
// ===== library types =====

// folder: NN_types

TYPE "scaler_type"
   STRUCT
      data_min : Array[1.."MAX_NO_NEURONS_PER_LAYER"] of Real;
      data_max : Array[1.."MAX_NO_NEURONS_PER_LAYER"] of Real;
      range_min : Real;
      range_max : Real;
   END_STRUCT;
END_TYPE

TYPE "NN_config_type"
   STRUCT
      NumLayers : Int := 5;
      NeuronPerLayer : Array[1.."MAX_NO_LAYERS"] of Int;
      ActivationFunction : Array[1.."MAX_NO_LAYERS"] of Int;   // 1=sigmoid; 2=ReLU; 3= Tanh; 4=LeakyReLU; 5= Softmax
      neuron : Array[1.."MAX_NO_LAYERS", 1.."MAX_NO_NEURONS_PER_LAYER"] of Real;
      weight : Array[1.."MAX_NO_LAYERS", 1.."MAX_NO_NEURONS_PER_LAYER", 1.."MAX_NO_NEURONS_PER_LAYER"] of Real;
      bias : Array[1.."MAX_NO_LAYERS", 1.."MAX_NO_NEURONS_PER_LAYER"] of Real;
      scalerParam : "scaler_type";
   END_STRUCT;
   // NeuronPerLayer[1] := 7;
   // NeuronPerLayer[2] := 128;
   // NeuronPerLayer[3] := 64;
   // NeuronPerLayer[4] := 32;
   // NeuronPerLayer[5] := 6;
   // ActivationFunction[1] := 2;
   // ActivationFunction[2] := 2;
   // ActivationFunction[3] := 2;
   // ActivationFunction[4] := 2;
   // ActivationFunction[5] := 5;
END_TYPE

// folder: NN

FUNCTION_BLOCK "NN_MLP"   // FB19000, SCL
{ S7_Optimized_Access := 'TRUE' }
VERSION : 0.1
   VAR_INPUT
      predict : Bool;
      contPredict : Bool;
      X : Array[1.."MAX_NO_NEURONS_PER_LAYER"] of Real;
   END_VAR
   VAR_OUTPUT
      done : Bool;
      busy : Bool;
      probability : Array[1.."MAX_NO_NEURONS_PER_LAYER"] of Real;
   END_VAR
   VAR_IN_OUT
      config : "NN_config_type";
   END_VAR
   VAR
      X_scaled : Array[1.."MAX_NO_NEURONS_PER_LAYER"] of Real;
      p : Int;
      n : Int;
      neuron_L : Int;
      "neuron_L+1" : Int;
      k : Int;
      layer_L : Int;
      s1 : Int;
      s2 : Int;
      S3 : Int;
      S4 : Int;
      statSumEXP : Real;
      statEXP : Array[1..6] of Real;
      statSoftmax : Array[1..6] of Real;
      statTotalSum : Real;
      predictRT : R_TRIG;
      statMemRuntime : LReal;
      timeExecution : LReal;
   END_VAR
BEGIN
   #predictRT(CLK := #predict);
   IF #predictRT.Q OR #contPredict THEN
       #timeExecution:= RUNTIME(#statMemRuntime);

       #done := FALSE;
       #busy := TRUE;

       REGION Entradas dos dados do processo  
           // normalização dos valores de entrada da rede neural. Dados retirados da função MinMaxScaler utilizada no tratamento dos dados da aplicação em python
           #config.scalerParam.data_min[1] := 295.3;
           #config.scalerParam.data_min[2] := 305.7;
           #config.scalerParam.data_min[3] := 1168.0;
           #config.scalerParam.data_min[4] := 3.8;
           #config.scalerParam.data_min[5] := 0.0;
           #config.scalerParam.data_min[6] := 0.0;
           #config.scalerParam.data_min[7] := 0.0;

           #config.scalerParam.data_max[1] := 304.5;
           #config.scalerParam.data_max[2] := 313.8;
           #config.scalerParam.data_max[3] := 2886.0;
           #config.scalerParam.data_max[4] := 76.6;
           #config.scalerParam.data_max[5] := 253.0;
           #config.scalerParam.data_max[6] := 1.0;
           #config.scalerParam.data_max[7] := 1.0;

           #config.scalerParam.range_min := -1.0;
           #config.scalerParam.range_max := 1.0;

           FOR #n := 1 TO #config.NeuronPerLayer[1] DO
               #X_scaled[#n] := (#X[#n] - #config.scalerParam.data_min[#n]) /
               (#config.scalerParam.data_max[#n] - #config.scalerParam.data_min[#n]) *
               (#config.scalerParam.range_max - #config.scalerParam.range_min) +
               #config.scalerParam.range_min;
           END_FOR;

       END_REGION

       REGION Transferencia dados de entrada para a primeira camada da rede neural    
           FOR #"neuron_L" := 1 TO #config.NeuronPerLayer[1] DO
               #config.neuron[1, #"neuron_L"] := #X_scaled[#"neuron_L"];
           END_FOR;
       END_REGION

       REGION Forward

           FOR #layer_L := 1 TO #config.NumLayers - 1 DO
               FOR #"neuron_L+1" := 1 TO #config.NeuronPerLayer[#layer_L + 1] DO
                   #config.neuron[#layer_L + 1, #"neuron_L+1"] := 0;
                   FOR #"neuron_L" := 1 TO #config.NeuronPerLayer[#layer_L] DO
                       #config.neuron[#layer_L + 1, #"neuron_L+1"] := #config.neuron[#layer_L + 1, #"neuron_L+1"] +
                       (#config.neuron[#layer_L, #"neuron_L"] *
                       #config.weight[#layer_L, #"neuron_L+1", #"neuron_L"]);
                   END_FOR;
                   #config.neuron[#layer_L + 1, #"neuron_L+1"] := #config.neuron[#layer_L + 1, #"neuron_L+1"] + #config.bias[#layer_L, #"neuron_L+1"];

                   CASE #config.ActivationFunction[#layer_L + 1] OF
                       1:
                           #config.neuron[#layer_L + 1, #"neuron_L+1"] := 1.0 / (1.0 + EXP(- #config.neuron[#layer_L + 1, #"neuron_L+1"]));
                       2:
                           IF #config.neuron[#layer_L + 1, #"neuron_L+1"] <= 0.0 THEN
                               #config.neuron[#layer_L + 1, #"neuron_L+1"] := 0.0;
                           END_IF;
                       3:
                           #config.neuron[#layer_L + 1, #"neuron_L+1"] := (EXP(#config.neuron[#layer_L + 1, #"neuron_L+1"])
                           - EXP(- #config.neuron[#layer_L + 1, #"neuron_L+1"]))
                           / (EXP(#config.neuron[#layer_L + 1, #"neuron_L+1"])
                           + EXP(- #config.neuron[#layer_L + 1, #"neuron_L+1"]));
                       4:
                           IF #config.neuron[#layer_L + 1, #"neuron_L+1"] <= 0.0 THEN
                               #config.neuron[#layer_L + 1, #"neuron_L+1"] := "ALPHA" * #config.neuron[#layer_L + 1, #"neuron_L+1"];
                           END_IF;
                       5:
                           IF #layer_L = #config.NumLayers - 1 THEN
                               #statSumEXP := 0.0;
                               #statTotalSum := 0.0;
                               FOR #s1 := 1 TO #config.NeuronPerLayer[#layer_L + 1] BY 1 DO
                                   #statEXP[#s1] := EXP(#config.neuron[#layer_L + 1, #s1]);
                               END_FOR;
                               FOR #s2 := 1 TO #config.NeuronPerLayer[#layer_L + 1] BY 1 DO
                                   #statSumEXP := #statSumEXP + #statEXP[#s2];
                               END_FOR;
                               FOR #S3 := 1 TO #config.NeuronPerLayer[#layer_L + 1] BY 1 DO
                                   #statSoftmax[#S3] := #statEXP[#S3] / #statSumEXP;
                               END_FOR;
                               FOR #S4 := 1 TO #config.NeuronPerLayer[#layer_L + 1] BY 1 DO
                                   #statTotalSum := #statTotalSum + #statSoftmax[#S4];
                               END_FOR;
                           END_IF;
                   END_CASE;
               END_FOR;
           END_FOR;
           FOR #p := 1 TO #config.NeuronPerLayer["MAX_NO_LAYERS"] DO
               #probability[#p] := #statSoftmax[#p] * 100.0;
           END_FOR;
       END_REGION

           #done := TRUE;
           #busy := FALSE;
           #timeExecution := RUNTIME(#statMemRuntime);

       END_IF;
END_FUNCTION_BLOCK

// ===== library: MasterCopy "NN_GetWeightsAndBias" =====

// folder: NN

FUNCTION_BLOCK "NN_GetWeightsAndBias"   // FB19002, SCL
{ S7_Optimized_Access := 'TRUE' }
VERSION : 0.1
   VAR
      index_j : Int;
      index_i : Int;
   END_VAR
BEGIN

   //A transferencia dos valores dos pesos e dos biases ocorre via Snap7 que permite apenas o uso de data blocks (DB's) não otimizados.
   //Os DBs não otimizados tem memória restrita a 65536 bytes. Como cada valor de peso ocupa 4 bytes de memória, por ser do tipo real, seria possivel armazenar no máximo
   //16 384 parametros o que pode restringir o uso de redes com mais camadas e/ou neuronios. 
   //Para generalizar o uso do código abaixo de forma a causar menos interferencia caso outras arquiteturas de rede devam ser utilizadas, será utilizado um DB
   //otimizado que possui maior capacidade para o armazenamento dos valores de pesos, bias e configurações.

   REGION Transferencia de dados do DB não otimizado para DB otimizado

       FOR #index_i := 1 TO 128 DO
           FOR #index_j := 1 TO 7 DO
               "NN_Config".weight[1, #index_i, #index_j] :="NN_Parameters_weight_bias".weight_1[#index_i, #index_j];
           END_FOR;
           "NN_Config".bias[1, #index_i] := "NN_Parameters_weight_bias".bias_1[#index_i];
       END_FOR;

       FOR #index_i := 1 TO 64 DO
           FOR #index_j := 1 TO 128 DO
               "NN_Config".weight[2, #index_i, #index_j] := "NN_Parameters_weight_bias".weight_2[#index_i, #index_j];
           END_FOR;
           "NN_Config".bias[2, #index_i] := "NN_Parameters_weight_bias".bias_2[#index_i];
       END_FOR;

       FOR #index_i := 1 TO 32 DO
           FOR #index_j := 1 TO 64 DO
               "NN_Config".weight[3, #index_i, #index_j] := "NN_Parameters_weight_bias".weight_3[#index_i, #index_j];
           END_FOR;
           "NN_Config".bias[3, #index_i] := "NN_Parameters_weight_bias".bias_3[#index_i];
       END_FOR;

       FOR #index_i := 1 TO 6 DO
           FOR #index_j := 1 TO 32 DO
               "NN_Config".weight[4, #index_i, #index_j] := "NN_Parameters_weight_bias".weight_4[#index_i, #index_j];
           END_FOR;
           "NN_Config".bias[4, #index_i] := "NN_Parameters_weight_bias".bias_4[#index_i];
       END_FOR;

   END_REGION
END_FUNCTION_BLOCK

// ===== library: MasterCopy "NN_Config" =====

// folder: NN

DATA_BLOCK "NN_Config"   // DB19000
{ S7_Optimized_Access := 'TRUE' }
VERSION : 0.1
BEGIN
END_DATA_BLOCK

// ===== library: MasterCopy "NN_LearnableBias" =====

// folder: NN

DATA_BLOCK "NN_LearnableBias"   // DB19002
{ S7_Optimized_Access := 'FALSE' }
VERSION : 0.1
   VAR
      layer_1 : "layer1_bias_type";
      layer_2 : "layer2_bias_type";
      layer_3 : "layer3_bias_type";
      layer_4 : "layer4_bias_type";
   END_VAR
BEGIN
END_DATA_BLOCK

// ===== library: MasterCopy "NN_LearnableWeights" =====

// folder: NN

DATA_BLOCK "NN_LearnableWeights"   // DB19003
{ S7_Optimized_Access := 'FALSE' }
VERSION : 0.1
   VAR
      layer_1 : "layer1_weight_type";
      layer_2 : "layer2_weight_type";
      layer_3 : "layer3_weight_type";
      layer_4 : "layer4_weight_type";
   END_VAR
BEGIN
END_DATA_BLOCK

// ===== library: MasterCopy "NN_Parameters_weight_bias" =====

// folder: NN

DATA_BLOCK "NN_Parameters_weight_bias"   // DB19005
{ S7_Optimized_Access := 'FALSE' }
VERSION : 0.1
   VAR
      weight_1 : Array[1..128, 1..7] of Real;
      bias_1 : Array[1..128] of Real;
      weight_2 : Array[1..64, 1..128] of Real;
      bias_2 : Array[1..64] of Real;
      weight_3 : Array[1..32, 1..64] of Real;
      bias_3 : Array[1..32] of Real;
      weight_4 : Array[1..6, 1..32] of Real;
      bias_4 : Array[1..6] of Real;
   END_VAR
BEGIN
END_DATA_BLOCK

// ===== library: MasterCopy "NN_ScalerData" =====

// folder: NN

DATA_BLOCK "NN_ScalerData"   // DB19001
{ S7_Optimized_Access := 'FALSE' }
VERSION : 0.1
   VAR
      data_min : Array[1..7] of Real;
      data_max : Array[1..7] of Real;
      range_min : Real;
      range_max : Real;
   END_VAR
BEGIN
END_DATA_BLOCK

// ===== library: MasterCopy "NN_MLP" =====

// folder: NN

FUNCTION_BLOCK "NN_MLP"   // FB19000, SCL
{ S7_Optimized_Access := 'TRUE' }
VERSION : 0.1
   VAR_INPUT
      predict : Bool;
      contPredict : Bool;
      X : Array[1.."MAX_NO_NEURONS_PER_LAYER"] of Real;
   END_VAR
   VAR_OUTPUT
      done : Bool;
      busy : Bool;
      probability : Array[1.."MAX_NO_NEURONS_PER_LAYER"] of Real;
   END_VAR
   VAR_IN_OUT
      config : "NN_config_type";
   END_VAR
   VAR
      X_scaled : Array[1.."MAX_NO_NEURONS_PER_LAYER"] of Real;
      p : Int;
      n : Int;
      neuron_L : Int;
      "neuron_L+1" : Int;
      k : Int;
      layer_L : Int;
      s1 : Int;
      s2 : Int;
      S3 : Int;
      S4 : Int;
      statSumEXP : Real;
      statEXP : Array[1..6] of Real;
      statSoftmax : Array[1..6] of Real;
      statTotalSum : Real;
      predictRT : R_TRIG;
      statMemRuntime : LReal;
      timeExecution : LReal;
   END_VAR
BEGIN
   #predictRT(CLK := #predict);
   IF #predictRT.Q OR #contPredict THEN
       #timeExecution:= RUNTIME(#statMemRuntime);

       #done := FALSE;
       #busy := TRUE;

       REGION Entradas dos dados do processo  
           // normalização dos valores de entrada da rede neural. Dados retirados da função MinMaxScaler utilizada no tratamento dos dados da aplicação em python
           #config.scalerParam.data_min[1] := 295.3;
           #config.scalerParam.data_min[2] := 305.7;
           #config.scalerParam.data_min[3] := 1168.0;
           #config.scalerParam.data_min[4] := 3.8;
           #config.scalerParam.data_min[5] := 0.0;
           #config.scalerParam.data_min[6] := 0.0;
           #config.scalerParam.data_min[7] := 0.0;

           #config.scalerParam.data_max[1] := 304.5;
           #config.scalerParam.data_max[2] := 313.8;
           #config.scalerParam.data_max[3] := 2886.0;
           #config.scalerParam.data_max[4] := 76.6;
           #config.scalerParam.data_max[5] := 253.0;
           #config.scalerParam.data_max[6] := 1.0;
           #config.scalerParam.data_max[7] := 1.0;

           #config.scalerParam.range_min := -1.0;
           #config.scalerParam.range_max := 1.0;

           FOR #n := 1 TO #config.NeuronPerLayer[1] DO
               #X_scaled[#n] := (#X[#n] - #config.scalerParam.data_min[#n]) /
               (#config.scalerParam.data_max[#n] - #config.scalerParam.data_min[#n]) *
               (#config.scalerParam.range_max - #config.scalerParam.range_min) +
               #config.scalerParam.range_min;
           END_FOR;

       END_REGION

       REGION Transferencia dados de entrada para a primeira camada da rede neural    
           FOR #"neuron_L" := 1 TO #config.NeuronPerLayer[1] DO
               #config.neuron[1, #"neuron_L"] := #X_scaled[#"neuron_L"];
           END_FOR;
       END_REGION

       REGION Forward

           FOR #layer_L := 1 TO #config.NumLayers - 1 DO
               FOR #"neuron_L+1" := 1 TO #config.NeuronPerLayer[#layer_L + 1] DO
                   #config.neuron[#layer_L + 1, #"neuron_L+1"] := 0;
                   FOR #"neuron_L" := 1 TO #config.NeuronPerLayer[#layer_L] DO
                       #config.neuron[#layer_L + 1, #"neuron_L+1"] := #config.neuron[#layer_L + 1, #"neuron_L+1"] +
                       (#config.neuron[#layer_L, #"neuron_L"] *
                       #config.weight[#layer_L, #"neuron_L+1", #"neuron_L"]);
                   END_FOR;
                   #config.neuron[#layer_L + 1, #"neuron_L+1"] := #config.neuron[#layer_L + 1, #"neuron_L+1"] + #config.bias[#layer_L, #"neuron_L+1"];

                   CASE #config.ActivationFunction[#layer_L + 1] OF
                       1:
                           #config.neuron[#layer_L + 1, #"neuron_L+1"] := 1.0 / (1.0 + EXP(- #config.neuron[#layer_L + 1, #"neuron_L+1"]));
                       2:
                           IF #config.neuron[#layer_L + 1, #"neuron_L+1"] <= 0.0 THEN
                               #config.neuron[#layer_L + 1, #"neuron_L+1"] := 0.0;
                           END_IF;
                       3:
                           #config.neuron[#layer_L + 1, #"neuron_L+1"] := (EXP(#config.neuron[#layer_L + 1, #"neuron_L+1"])
                           - EXP(- #config.neuron[#layer_L + 1, #"neuron_L+1"]))
                           / (EXP(#config.neuron[#layer_L + 1, #"neuron_L+1"])
                           + EXP(- #config.neuron[#layer_L + 1, #"neuron_L+1"]));
                       4:
                           IF #config.neuron[#layer_L + 1, #"neuron_L+1"] <= 0.0 THEN
                               #config.neuron[#layer_L + 1, #"neuron_L+1"] := "ALPHA" * #config.neuron[#layer_L + 1, #"neuron_L+1"];
                           END_IF;
                       5:
                           IF #layer_L = #config.NumLayers - 1 THEN
                               #statSumEXP := 0.0;
                               #statTotalSum := 0.0;
                               FOR #s1 := 1 TO #config.NeuronPerLayer[#layer_L + 1] BY 1 DO
                                   #statEXP[#s1] := EXP(#config.neuron[#layer_L + 1, #s1]);
                               END_FOR;
                               FOR #s2 := 1 TO #config.NeuronPerLayer[#layer_L + 1] BY 1 DO
                                   #statSumEXP := #statSumEXP + #statEXP[#s2];
                               END_FOR;
                               FOR #S3 := 1 TO #config.NeuronPerLayer[#layer_L + 1] BY 1 DO
                                   #statSoftmax[#S3] := #statEXP[#S3] / #statSumEXP;
                               END_FOR;
                               FOR #S4 := 1 TO #config.NeuronPerLayer[#layer_L + 1] BY 1 DO
                                   #statTotalSum := #statTotalSum + #statSoftmax[#S4];
                               END_FOR;
                           END_IF;
                   END_CASE;
               END_FOR;
           END_FOR;
           FOR #p := 1 TO #config.NeuronPerLayer["MAX_NO_LAYERS"] DO
               #probability[#p] := #statSoftmax[#p] * 100.0;
           END_FOR;
       END_REGION

           #done := TRUE;
           #busy := FALSE;
           #timeExecution := RUNTIME(#statMemRuntime);

       END_IF;
END_FUNCTION_BLOCK